// TIA Portal V17 export
// export: Created 2023-04-06T14:59:51.4519566Z, ExportSetting None, DisplayName Totally Integrated Automation Portal, DisplayVersion V17 Update 4, DisplayName TIA Portal Openness, DisplayVersion V17 Update 4, DisplayName TIA Portal Version Control Interface, DisplayVersion V17, DisplayName STEP 7 Professional, DisplayVersion V17 Update 4, DisplayName STEP 7 Safety, DisplayVersion V17, DisplayName WinCC Advanced / Unified PC, DisplayVersion V17 Update 4
DATA_BLOCK "SETTINGS"   // DB26
{ S7_Optimized_Access := 'FALSE' }
// stored: AutoNumber false
   VAR RETAIN
      PIT_33302 : Struct   // COMPRESSOR SUCTION PRESSURE
         RANGE_L : Real := 0.0;
         RANGE_H : Real := 24.0;
         SP_LL : Real := -100.0;
         SP_L : Real := -100.0;
         SP_H : Real := 124.0;
         SP_HH : Real := 124.0;
      END_STRUCT;
      PIT_33303 : Struct   // LUBE OIL SEPARATOR OUTLET PRESSURE
         RANGE_L : Real := 0.0;
         RANGE_H : Real := 24.0;
         SP_LL : Real := -100.0;
         SP_L : Real := -100.0;
         SP_H : Real := 124.0;
         SP_HH : Real := 124.0;
      END_STRUCT;
      LIT_33304 : Struct   // CONDENSER LEVEL
         RANGE_L : Real := 0.0;
         RANGE_H : Real := 100.0;
         SP_LL : Real := -100.0;
         SP_L : Real := -100.0;
         SP_H : Real := 200.0;
         SP_HH : Real := 200.0;
      END_STRUCT;
      PIT_33301 : Struct   // COMPRESSOR SUCTION PRESSURE
         RANGE_L : Real := 0.0;
         RANGE_H : Real := 24.0;
         SP_LL : Real := -100.0;
         SP_L : Real := -100.0;
         SP_H : Real := 124.0;
         SP_HH : Real := 124.0;
      END_STRUCT;
      TT_33302 : Struct   // LUBE OIL SEPARATOR OUTLET TEMPERATURE
         RANGE_L : Real := 0.0;
         RANGE_H : Real := 150.0;
         SP_LL : Real := -100.0;
         SP_L : Real := -100.0;
         SP_H : Real := 250.0;
         SP_HH : Real := 250.0;
      END_STRUCT;
      PIT_33304 : Struct   // LUBE OIL SEPARATOR OUTLET PRESSURE
         RANGE_L : Real := 0.0;
         RANGE_H : Real := 24.0;
         SP_LL : Real := -100.0;
         SP_L : Real := -100.0;
         SP_H : Real := 124.0;
         SP_HH : Real := 124.0;
      END_STRUCT;
      PDIT_33305 : Struct   // OIL DIFFERENTIAL PRESSURE
         RANGE_L : Real := 0.0;
         RANGE_H : Real := 6.0;
         SP_LL : Real := -100.0;
         SP_L : Real := -100.0;
         SP_H : Real := 106.0;
         SP_HH : Real := 106.0;
      END_STRUCT;
      TT_33303 : Struct   // OIL TEMPERATURE
         RANGE_L : Real := 0.0;
         RANGE_H : Real := 150.0;
         SP_LL : Real := -100.0;
         SP_L : Real := -100.0;
         SP_H : Real := 250.0;
         SP_HH : Real := 250.0;
      END_STRUCT;
      PDIT_33309 : Struct   // OIL FILTER DIFFERENTIAL PRESSURE
         RANGE_L : Real := 0.0;
         RANGE_H : Real := 1.0;
         SP_LL : Real := -100.0;
         SP_L : Real := -100.0;
         SP_H : Real := 101.0;
         SP_HH : Real := 101.0;
      END_STRUCT;
      PIT_33311 : Struct   // ECONOMIZER PRESSURE
         RANGE_L : Real := 0.0;
         RANGE_H : Real := 24.0;
         SP_LL : Real := -100.0;
         SP_L : Real := -100.0;
         SP_H : Real := 124.0;
         SP_HH : Real := 124.0;
      END_STRUCT;
      LIT_33305 : Struct   // ECONOMIZER LEVEL
         RANGE_L : Real := 0.0;
         RANGE_H : Real := 100.0;
         SP_LL : Real := -100.0;
         SP_L : Real := -100.0;
         SP_H : Real := 200.0;
         SP_HH : Real := 200.0;
      END_STRUCT;
      LIT_33309 : Struct   // KO DRUM LEVEL
         RANGE_L : Real := 0.0;
         RANGE_H : Real := 100.0;
         SP_LL : Real := -100.0;
         SP_L : Real := -100.0;
         SP_H : Real := 200.0;
         SP_HH : Real := 200.0;
      END_STRUCT;
      PIT_33315 : Struct   // LUBE OIL RECOVERY LINE PRESSURE
         RANGE_L : Real := 0.0;
         RANGE_H : Real := 24.0;
         SP_LL : Real := -100.0;
         SP_L : Real := -100.0;
         SP_H : Real := 124.0;
         SP_HH : Real := 124.0;
      END_STRUCT;
      LIT_33302 : Struct   // OIL SEPARATOR LEVEL
         RANGE_L : Real := 0.0;
         RANGE_H : Real := 100.0;
         SP_LL : Real := -100.0;
         SP_L : Real := -100.0;
         SP_H : Real := 200.0;
         SP_HH : Real := 200.0;
      END_STRUCT;
      FIT_33303 : Struct   // SEAL NITROGEN FLOW
         RANGE_L : Real := 0.0;
         RANGE_H : Real := 100.0;
         SP_LL : Real := -100.0;
         SP_L : Real := -100.0;
         SP_H : Real := 200.0;
         SP_HH : Real := 200.0;
      END_STRUCT;
      LIT_33311 : Struct   // COMPRESSOR SEAL POT LEVEL
         RANGE_L : Real := 0.0;
         RANGE_H : Real := 100.0;
         SP_LL : Real := -100.0;
         SP_L : Real := -100.0;
         SP_H : Real := 200.0;
         SP_HH : Real := 200.0;
      END_STRUCT;
      LIT_33310 : Struct   // OIL PUMP A SEAL POT LEVEL
         RANGE_L : Real := 0.0;
         RANGE_H : Real := 100.0;
         SP_LL : Real := -100.0;
         SP_L : Real := -100.0;
         SP_H : Real := 200.0;
         SP_HH : Real := 200.0;
      END_STRUCT;
      LIT_33312 : Struct   // OIL PUMP B SEAL POT LEVEL
         RANGE_L : Real := 0.0;
         RANGE_H : Real := 100.0;
         SP_LL : Real := -100.0;
         SP_L : Real := -100.0;
         SP_H : Real := 200.0;
         SP_HH : Real := 200.0;
      END_STRUCT;
      PIT_33314 : Struct   // OIL PUMP A SEAL POT PRESSURE
         RANGE_L : Real := 0.0;
         RANGE_H : Real := 100.0;
         SP_LL : Real := -100.0;
         SP_L : Real := -100.0;
         SP_H : Real := 200.0;
         SP_HH : Real := 200.0;
      END_STRUCT;
      PIT_33316 : Struct   // OIL PUMP B SEAL POT PRESSURE
         RANGE_L : Real := 0.0;
         RANGE_H : Real := 100.0;
         SP_LL : Real := -100.0;
         SP_L : Real := -100.0;
         SP_H : Real := 200.0;
         SP_HH : Real := 200.0;
      END_STRUCT;
      TT_33311 : Struct   // OIL SEPARATOR TEMPERATURE
         RANGE_L : Real := 0.0;
         RANGE_H : Real := 150.0;
         SP_LL : Real := -100.0;
         SP_L : Real := -100.0;
         SP_H : Real := 250.0;
         SP_HH : Real := 250.0;
      END_STRUCT;
      PIT_33313 : Struct   // COMPRESSOR SEAL POT PRESSURE
         RANGE_L : Real := 0.0;
         RANGE_H : Real := 100.0;
         SP_LL : Real := -100.0;
         SP_L : Real := -100.0;
         SP_H : Real := 200.0;
         SP_HH : Real := 200.0;
      END_STRUCT;
      II_33301 : Struct   // COMPRESSOR MAIN MOTOR CURRENT
         RANGE_L : Real := 0.0;
         RANGE_H : Real := 100.0;
         SP_LL : Real := -100.0;
         SP_L : Real := -100.0;
         SP_H : Real := 200.0;
         SP_HH : Real := 200.0;
      END_STRUCT;
      ZT_33302 : Struct   // SLIDE VALVE POSITION
         RANGE_L : Real := 0.0;
         RANGE_H : Real := 100.0;
         SP_LL : Real := -100.0;
         SP_L : Real := -100.0;
         SP_H : Real := 200.0;
         SP_HH : Real := 200.0;
      END_STRUCT;
   END_VAR
BEGIN
END_DATA_BLOCK
